{attribute 'Tc2GvlVarNames'}
VAR_GLOBAL
	fbCheckArrayBounds: FB_CheckArrayBounds;

	fbCheckDivRealInfo: FB_CheckDivRealInfo;
END_VAR

(* stored: Version 1.1.0.1, ProductVersion 3.1.4024.12
   GVL Globale_Variablen: Id {48a97b99-07a8-4b24-87e0-dba2f262fceb} *)
